// TIA Portal V17 export
// export: Created 2024-09-02T12:50:34.3207052Z, ExportSetting WithDefaults, DisplayName Totally Integrated Automation Portal, DisplayVersion V17, DisplayName TIA Portal Openness, DisplayVersion V17, DisplayName TIA Portal Version Control Interface, DisplayVersion V17, DisplayName STEP 7 Professional, DisplayVersion V17, DisplayName STEP 7 Safety, DisplayVersion V17, DisplayName WinCC Professional, DisplayVersion V17
TYPE "typ_MobyTAFDaten"
// stored: IsFailsafeCompliant false
   STRUCT
      Kopfdaten : Struct   // Kopfdaten / Head data
         GDAT { S7_SetPoint := 'True'} : "typ_General";   // Grunddaten / Basic Data
      END_STRUCT;
      Festbereich : Struct   // Festbereich / Fixed area
         KEY { S7_SetPoint := 'True'} : "typ_Key";   // Keydaten / key data
         PRG_TAF { S7_SetPoint := 'True'} : Array[1..8] of "typ_Arbeitsprg";   // Arbeitsprogramme / Work program
         STATUS_TAF : Array[1..768] of Byte;   // TAF Status / TAF Status
      END_STRUCT;
      Flexbereich : Struct   // Flexbereich / Flex area
         ANBAUTEILE_TAF { S7_SetPoint := 'True'} : Array[1..8] of "typ_AnbauteilVorg";   // Anbauteile / Attachment parts
         MELDEBYTE_TAF_MIT { S7_SetPoint := 'True'} : Array[1..8] of "typ_Einzelmeldung";   // Meldekontrolle mit Nacharbeit / Reporting control with reworking
         MELDEBYTE_TAF_OHNE { S7_SetPoint := 'True'} : Array[1..8] of "typ_Einzelmeldung";   // Meldekontrolle ohne Nacharbeit / Reporting control without reworking
         MELDEBYTE_TAF_NOK { S7_SetPoint := 'True'} : Array[1..8] of "typ_Einzelmeldung";
         DMC_TAF { ExternalWritable := 'False'; S7_SetPoint := 'True'} : Array[1..8] of "typ_MobyDMCTaf";   // DMC Ist Daten / DMC Actual data
      END_STRUCT;
      Anwender : Struct   // Freikonfigurierte Daten / Configured data
         D1 : Array[1..100] of Byte;   // Bereich kann erweitert werden / Range can be extended
         D2 : Array[1..100] of Byte;   // Bereich kann erweitert werden / Range can be extended
         D3 : Array[1..100] of Byte;   // Bereich kann erweitert werden / Range can be extended
         D4 : Array[1..100] of Byte;   // Bereich kann erweitert werden / Range can be extended
      END_STRUCT;
      QDaten { S7_SetPoint := 'True'} : Array[1..50] of "typ_QDS";   // QDaten / Qdata
      TAF : Struct
         Freigabe : Array[1..8] of Bool;
         Abwahl : Array[1..8] of Bool;
         Quali : Array[1..8] of Struct   // TAF
            QDaten { S7_SetPoint := 'True'} : Array[1..32] of "typ_QDS";   // QDaten / Qdata
         END_STRUCT;
         DMC { ExternalWritable := 'False'; S7_SetPoint := 'True'} : Array[1..8] of "typ_MobyDMCTaf";   // DMC Ist Daten / DMC Actual data
      END_STRUCT;
   END_STRUCT;
END_TYPE
